// TIA Portal V17 export
// export: Created 2024-09-02T12:50:32.52467Z, ExportSetting WithDefaults, DisplayName Totally Integrated Automation Portal, DisplayVersion V17, DisplayName TIA Portal Openness, DisplayVersion V17, DisplayName TIA Portal Version Control Interface, DisplayVersion V17, DisplayName STEP 7 Professional, DisplayVersion V17, DisplayName STEP 7 Safety, DisplayVersion V17, DisplayName WinCC Professional, DisplayVersion V17
TYPE "Omron_Output"
// stored: IsFailsafeCompliant false
   STRUCT
      "Controle_Output(2Words)" : Struct
         Chanel0 : Struct
            Flg : Bool;
            Busy : Bool;
            Reserve_2 : Bool;
            "OR" : Bool;
            Run : Bool;
            Reserve_5 : Bool;
            Reserve_6 : Bool;
            Reserve_7 : Bool;
            XFlag : Bool;
            Xbusy : Bool;
            xWait : Bool;
            Reserve_11 : Bool;
            Reserve_12 : Bool;
            Reserve_13 : Bool;
            Reserve_14 : Bool;
            Err : Bool;
         END_STRUCT;
         Chanel1 : Struct
            Gate : Bool;
            Reserve_1 : Bool;
            Reserve_2 : Bool;
            Reserve_3 : Bool;
            Reserve_4 : Bool;
            Reserve_5 : Bool;
            Reserve_6 : Bool;
            Reserve_7 : Bool;
            Reserve_8 : Bool;
            Reserve_9 : Bool;
            Reserve_10 : Bool;
            Reserve_11 : Bool;
            Reserve_12 : Bool;
            Reserve_13 : Bool;
            Reserve_14 : Bool;
            Reserve_15 : Bool;
         END_STRUCT;
      END_STRUCT;
      "Command_Code(2Words)" : Struct
         Chanel2 : Word;
         Chanel3 : Word;
      END_STRUCT;
      "Response_Code(2Words)" : Struct
         Chanel4 : Struct
            Reserve_0 : Bool;
            Reserve_1 : Bool;
            Reserve_2 : Bool;
            Reserve_3 : Bool;
            Reserve_4 : Bool;
            Reserve_5 : Bool;
            Reserve_6 : Bool;
            Reserve_7 : Bool;
            Reserve_8 : Bool;
            Reserve_9 : Bool;
            Reserve_10 : Bool;
            Reserve_11 : Bool;
            Reserve_12 : Bool;
            Reserve_13 : Bool;
            Reserve_14 : Bool;
            Reserve_15 : Bool;
         END_STRUCT;
         Chanel5 : Struct
            Reserve_0 : Bool;
            Reserve_1 : Bool;
            Reserve_2 : Bool;
            Reserve_3 : Bool;
            Reserve_4 : Bool;
            Reserve_5 : Bool;
            Reserve_6 : Bool;
            Reserve_7 : Bool;
            Reserve_8 : Bool;
            Reserve_9 : Bool;
            Reserve_10 : Bool;
            Reserve_11 : Bool;
            Reserve_12 : Bool;
            Reserve_13 : Bool;
            Reserve_14 : Bool;
            Reserve_15 : Bool;
         END_STRUCT;
      END_STRUCT;
      "Response_Data(2Words)" : Struct
         Chanel6 : Struct
            Reserve_0 : Bool;
            Reserve_1 : Bool;
            Reserve_2 : Bool;
            Reserve_3 : Bool;
            Reserve_4 : Bool;
            Reserve_5 : Bool;
            Reserve_6 : Bool;
            Reserve_7 : Bool;
            Reserve_8 : Bool;
            Reserve_9 : Bool;
            Reserve_10 : Bool;
            Reserve_11 : Bool;
            Reserve_12 : Bool;
            Reserve_13 : Bool;
            Reserve_14 : Bool;
            Reserve_15 : Bool;
         END_STRUCT;
         Chanel7 : Struct
            Reserve_0 : Bool;
            Reserve_1 : Bool;
            Reserve_2 : Bool;
            Reserve_3 : Bool;
            Reserve_4 : Bool;
            Reserve_5 : Bool;
            Reserve_6 : Bool;
            Reserve_7 : Bool;
            Reserve_8 : Bool;
            Reserve_9 : Bool;
            Reserve_10 : Bool;
            Reserve_11 : Bool;
            Reserve_12 : Bool;
            Reserve_13 : Bool;
            Reserve_14 : Bool;
            Reserve_15 : Bool;
         END_STRUCT;
      END_STRUCT;
      "Data0(2Words)" : Struct
         Chanel6 : Struct
            Reserve_0 : Bool;
            Reserve_1 : Bool;
            Reserve_2 : Bool;
            Reserve_3 : Bool;
            Reserve_4 : Bool;
            Reserve_5 : Bool;
            Reserve_6 : Bool;
            Reserve_7 : Bool;
            Reserve_8 : Bool;
            Reserve_9 : Bool;
            Reserve_10 : Bool;
            Reserve_11 : Bool;
            Reserve_12 : Bool;
            Reserve_13 : Bool;
            Reserve_14 : Bool;
            Reserve_15 : Bool;
         END_STRUCT;
         Chanel7 : Struct
            Reserve_0 : Bool;
            Reserve_1 : Bool;
            Reserve_2 : Bool;
            Reserve_3 : Bool;
            Reserve_4 : Bool;
            Reserve_5 : Bool;
            Reserve_6 : Bool;
            Reserve_7 : Bool;
            Reserve_8 : Bool;
            Reserve_9 : Bool;
            Reserve_10 : Bool;
            Reserve_11 : Bool;
            Reserve_12 : Bool;
            Reserve_13 : Bool;
            Reserve_14 : Bool;
            Reserve_15 : Bool;
         END_STRUCT;
      END_STRUCT;
   END_STRUCT;
END_TYPE
